VAR_GLOBAL
	hmiHeaderInstance	:	FB_HMIHeader;
	hmiHeaderInterface	:	HMIHeader;	
	hmiOperatingmodeInterface	:	HMIInterfaceOperatingMode;
	
	hmiAdsCommunicationInterfaceInstance	:	FB_ADSCommunicationStatus;
	hmiAdsCommunicationInterface	:	ADSCommunicationInterface;
	
	hmiMachineSectionInterface	:	MachineSectionHMIInterface;
	
	hmiEmitterInstances	:	ARRAY[0..0] OF STRING := [
														'FeedIn'
													];
	hmiConveyorInstances	:	ARRAY[0..5] OF STRING := [
															'FeedIn',
															'FeedIn StackerCrane',
															'FeedOut StackerCrane',
															'FeedOut Two meter',
															'FeedOut Curve',
															'FeedOut long'
														 ];
	hmiStackerCraneInstances	:	ARRAY[0..0] OF STRING := [
															'StackerCrane'
														 ];		
	hmiRFIDInstances	:	ARRAY[0..0] OF STRING := [
															'FeedIn StackerCrane'
														 ];
	hmiRemoverInstances	:	ARRAY[0..0] OF STRING := [
														'FeedOut'
													];
END_VAR

(* stored: Version 1.1.0.1
   GVL HMI: Id {42b8ab01-74f8-4d3b-9b14-9c080998c4d7} *)
